SUBAPPLICATION Uebung_210b_AR (* Standard IEC 61131-3 AI_FB_CTU (Adapter Version, Vorwärtszähler, INT) mit Terminal-Ausgabe (PHYS) *)
  (* Standard: 61131-3; Description: Copyright (c) 2026 Meisterschulen am Ostbahnhof This program and the accompanying materials are made available under the terms of the Eclipse Public License 2.0 which is available at https://www.eclipse.org/legal/epl-2.0/ SPDX-License-Identifier: EPL-2.0 *)
  (* Version 1.2, 2026-05-13, Franz Höpfinger, Meisterschulen am Ostbahnhof, Added AI_INT_TO_I init block connected to PV *)
  (* Version 1.1, 2026-04-21, Franz Höpfinger, Meisterschulen am Ostbahnhof, Added terminal output for counter value (PHYS) *)
  (* Version 1.0, 2026-04-21, Franz Höpfinger, Meisterschulen am Ostbahnhof, initial API and implementation (Adapter version) *)
  PACKAGE Uebungen;
  IMPORT Uebungen::const::UT::DefaultPool_Numeric::OutputNumber_N3_N;
  IMPORT logiBUS::io::DI::logiBUS_DI::Input_I1;
  IMPORT logiBUS::io::DI::logiBUS_DI::Input_I2;
  IMPORT logiBUS::io::DQ::logiBUS_DO::Output_Q1;
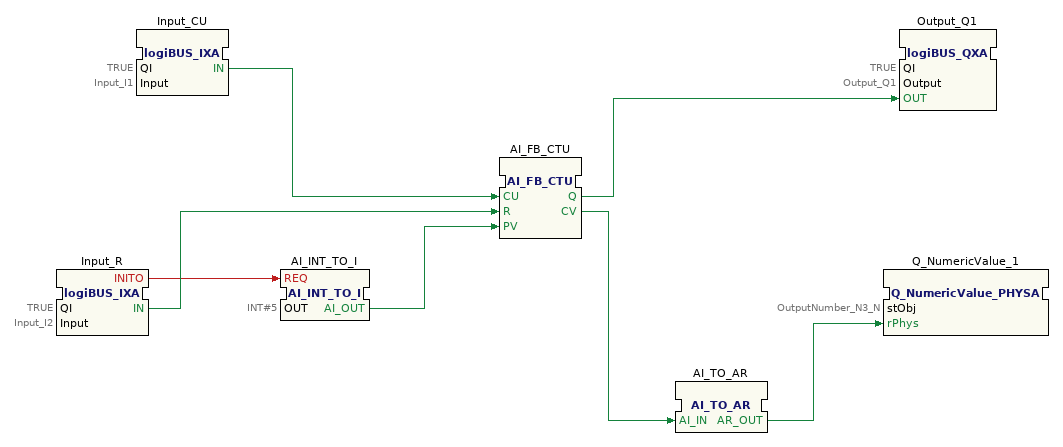
  (* hier sind negative Werte möglich ! *)
  (* hier gegebenenfalls einen AX_D_FF einbauen, damit die Events reduziert werden. *)
  FBS
    AI_FB_CTU : adapter::iec61131::counters::AI_FB_CTU;
    AI_INT_TO_I : adapter::conversion::unidirectional::AI_INT_TO_I(OUT := INT#5);
    Input_CU : logiBUS::io::DI::logiBUS_IXA(QI := TRUE, Input := Input_I1);
    Input_R : logiBUS::io::DI::logiBUS_IXA(QI := TRUE, Input := Input_I2);
    Output_Q1 : logiBUS::io::DQ::logiBUS_QXA(QI := TRUE, Output := Output_Q1);
    AI_TO_AR : adapter::conversion::unidirectional::AI_TO_AR;
    Q_NumericValue_1 : isobus::UT::Q::Q_NumericValue_PHYSA(stObj := OutputNumber_N3_N);
  END_FBS
  EVENT_CONNECTIONS
    Input_R.INITO TO AI_INT_TO_I.REQ;
  END_CONNECTIONS
  ADAPTER_CONNECTIONS
    Input_CU.IN TO AI_FB_CTU.CU;
    Input_R.IN TO AI_FB_CTU.R;
    AI_FB_CTU.Q TO Output_Q1.OUT;
    AI_FB_CTU.CV TO AI_TO_AR.AI_IN;
    AI_TO_AR.AR_OUT TO Q_NumericValue_1.rPhys;
    AI_INT_TO_I.AI_OUT TO AI_FB_CTU.PV;
  END_CONNECTIONS
END_SUBAPPLICATION
